# EPICS autosave request: GalilSup/Db/galil_userdef_records8.req
$(P)$(M)01_$(GS)_SP.VAL
$(P)$(M)02_$(GS)_SP.VAL
$(P)$(M)03_$(GS)_SP.VAL
$(P)$(M)04_$(GS)_SP.VAL
$(P)$(M)05_$(GS)_SP.VAL
$(P)$(M)06_$(GS)_SP.VAL
$(P)$(M)07_$(GS)_SP.VAL
$(P)$(M)08_$(GS)_SP.VAL
